TYPE AX5000_P_0800 :
STRUCT
	Digital_output_control_word:UINT;
END_STRUCT
END_TYPE

(* stored: Version 1.1.0.1, ProductVersion 3.1.4024.3
   DUT AX5000_P_0800: Id {7a215b8d-e21b-4458-a7d0-903e62955909} *)
